// TIA Portal V20 export
FUNCTION_BLOCK "FB_DigitalOutput"   // FB32, SCL
{ S7_Optimized_Access := 'TRUE' }
// stored: AutoNumber false, MemoryReserve 100, SetENOAutomatically false
   VAR_OUTPUT
      oHWStatus : Bool;
   END_VAR
   VAR
      sSWStatus { ExternalAccessible := 'False'; ExternalVisible := 'False'; ExternalWritable := 'False'} : Bool;
      sHWStatus { ExternalAccessible := 'False'; ExternalVisible := 'False'; ExternalWritable := 'False'} : Bool;
   END_VAR
BEGIN
   REGION Description header 
       //==================================================================================
       // POSALUX Swiss SA / (C) Copyright 2024
       //----------------------------------------------------------------------------------
       // Title: Fonction Sortie Numérique
       // Comment/Function: This function handles the state of a PLC digital output.
       //                   It updates the hardware output state based on the software
       //                   state and assigns this state to the PLC's physical output.
       // Author: Gowsigan SRITHARAN
       // Engineering: TIA Portal v17
       //----------------------------------------------------------------------------------
       // Change log table:
       // Version  | Date     | Expert in charge | Changes applied
       // ---------|----------|------------------|------------------------------------
       // 00.00.01 | 20250106 | GSR              | First released version
       // ==================================================================================
   END_REGION

   REGION Hardware State Update
       #sHWStatus := #sSWStatus;
   END_REGION

   REGION Physical Output Assignment
       #oHWStatus := #sHWStatus;
   END_REGION
END_FUNCTION_BLOCK
